FUNCTION F_Tollerance : BOOL
VAR_INPUT
	Variable: LREAL;
	reqValue: LREAL;

	Tollerance: LREAL;


END_VAR
VAR
END_VAR

IF Variable >= reqValue - Tollerance 
AND Variable <= reqValue + Tollerance
THEN;
	F_Tollerance:=TRUE;
ELSE;	
	F_Tollerance:=FALSE;
END_IF

END_FUNCTION

(* stored: Version 1.1.0.1, ProductVersion 3.1.4024.12
   POU F_Tollerance: Id {4fbf3e00-2e67-418e-a6c2-55110a601dae}, SpecialFunc None *)
